// Mitsubishi GX Works2 project: deng   PLC: FX1S

PROGRAM MAIN
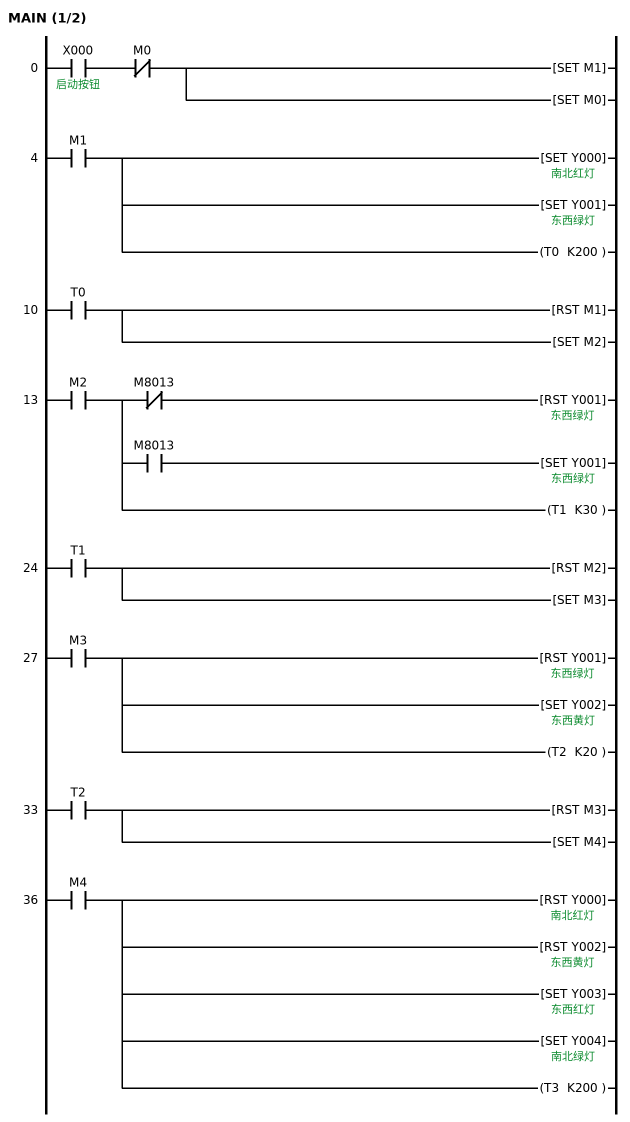
0     LD      X000  ; 启动按钮
      ANI     M0
      SET     M1
      SET     M0
4     LD      M1
      SET     Y000  ; 南北红灯
      SET     Y001  ; 东西绿灯
      OUT     T0 K200
10    LD      T0
      RST     M1
      SET     M2
13    LD      M2
      MPS
      ANI     M8013
      RST     Y001  ; 东西绿灯
      MRD
      AND     M8013
      SET     Y001  ; 东西绿灯
      MPP
      OUT     T1 K30
24    LD      T1
      RST     M2
      SET     M3
27    LD      M3
      RST     Y001  ; 东西绿灯
      SET     Y002  ; 东西黄灯
      OUT     T2 K20
33    LD      T2
      RST     M3
      SET     M4
36    LD      M4
      RST     Y000  ; 南北红灯
      RST     Y002  ; 东西黄灯
      SET     Y003  ; 东西红灯
      SET     Y004  ; 南北绿灯
      OUT     T3 K200
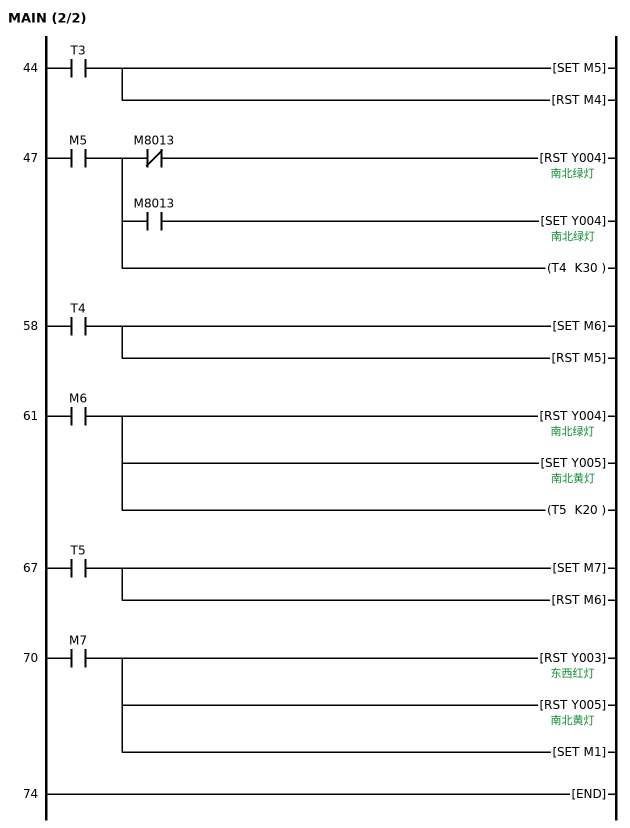
44    LD      T3
      SET     M5
      RST     M4
47    LD      M5
      MPS
      ANI     M8013
      RST     Y004  ; 南北绿灯
      MRD
      AND     M8013
      SET     Y004  ; 南北绿灯
      MPP
      OUT     T4 K30
58    LD      T4
      SET     M6
      RST     M5
61    LD      M6
      RST     Y004  ; 南北绿灯
      SET     Y005  ; 南北黄灯
      OUT     T5 K20
67    LD      T5
      SET     M7
      RST     M6
70    LD      M7
      RST     Y003  ; 东西红灯
      RST     Y005  ; 南北黄灯
      SET     M1
74    END
END_PROGRAM
